{attribute 'TcGenerated'}
{attribute 'no-analysis'}
{attribute 'linkalways'}
// This function has been automatically generated from the project information.
VAR_GLOBAL CONSTANT
    {attribute 'const_non_replaced'}
    stLibVersion_KFE_ARBITER : ST_LibVersion := (iMajor := 2, iMinor := 4, iBuild := 1, iRevision := 0, nFlags := 1, sVersion := '2.4.1');
END_VAR

(* stored: Version 1.1.0.1, ProductVersion 3.1.4022.18
   GVL Global_Version: Id {6fea7194-5f85-49a4-bba2-a8063801531c} *)
